FUNCTION_BLOCK CM_Sensor2State
VAR_INPUT
	PI_ManualMode : BOOL;
	PI_AutoMode : BOOL;
	
	PI_HMI_HAND : BOOL;
	PI_HMI_HAND_ON : BOOL;
	
	PI_Manual_ON : BOOL;
	PI_AutoHigh : BOOL;
	
	PI_AlarmHighEnable : BOOL;
	PI_AlarmLowEnable : BOOL;
	PI_Alarmdelay_H : DINT;
	PI_Alarmdelay_L : DINT;
	
	PI_Alarm_Condition_H : BOOL;
	PI_Alarm_Condition_L : BOOL;
	
	
	
END_VAR
VAR_OUTPUT
	PO_HMI_HAND : BOOL;
	PO_Manual : BOOL;
	PO_High : BOOL;
	
	PO_Alarm_H : BOOL;
	PO_Alarm_L : BOOL;
END_VAR
VAR
	Alarm_limit_Exceeded_H : BOOL;
	Alarm_limit_Exceeded_L : BOOL;
	
	prg_scan_H : DINT; // used for alarm delay
	prg_scan_L : DINT; // used for alarm delay
	
	Alarm_Ack_H : BOOL;
	Alarm_Ack_L : BOOL;
	
	alarmDelay_H : systemTimeDelay;
	alarmDelay_L : systemTimeDelay;
END_VAR
VAR_IN_OUT
	CM_UDT_CTRL : Udt_CM_Sensor2State;
	Plant_control : Udt_PlantControl;
END_VAR
VAR // added by the converter: edge detectors and wires of the graphical bodies
    _w1, _w2 : BOOL;
END_VAR

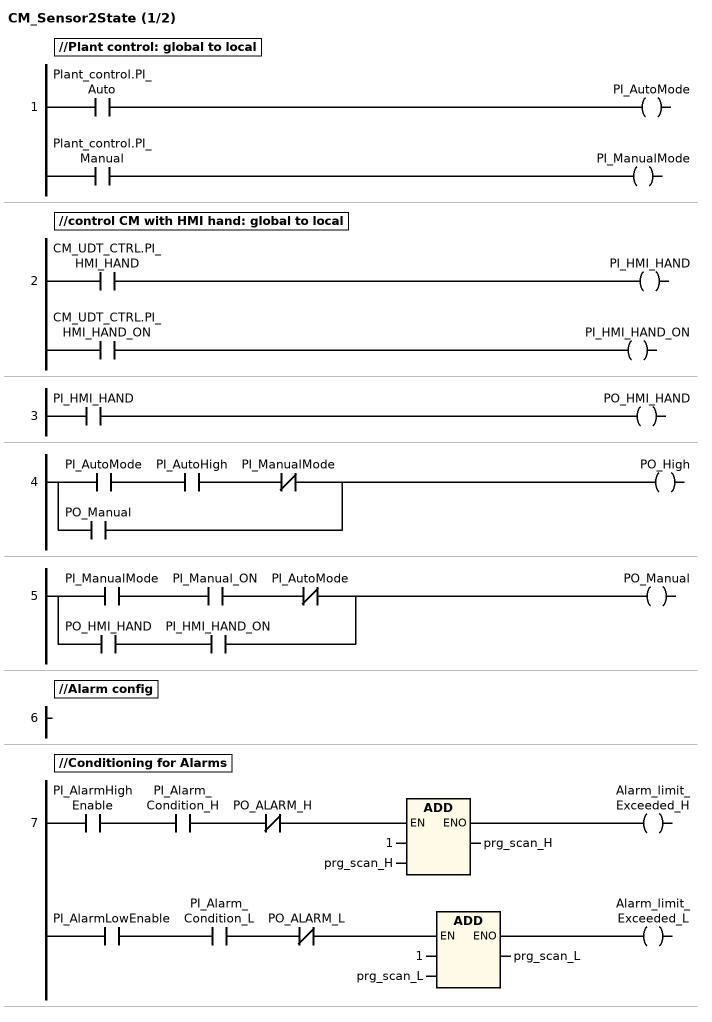
// NETWORK 1
// label: //Plant control: global to local
PI_AutoMode := Plant_control.PI_Auto;
PI_ManualMode := Plant_control.PI_Manual;

// NETWORK 2
// label: //control CM with HMI hand: global to local
PI_HMI_HAND := CM_UDT_CTRL.PI_HMI_HAND;
PI_HMI_HAND_ON := CM_UDT_CTRL.PI_HMI_HAND_ON;

// NETWORK 3
PO_HMI_HAND := PI_HMI_HAND;

// NETWORK 4
PO_High := PI_AutoMode AND PI_AutoHigh AND NOT PI_ManualMode OR PO_Manual;

// NETWORK 5
PO_Manual := PI_ManualMode AND PI_Manual_ON AND NOT PI_AutoMode OR PO_HMI_HAND AND PI_HMI_HAND_ON;

// NETWORK 6
// label: //Alarm config

// NETWORK 7
// label: //Conditioning for Alarms
_w1 := PI_AlarmHighEnable AND PI_Alarm_Condition_H AND NOT PO_ALARM_H;
IF _w1 THEN prg_scan_H := 1 + prg_scan_H; END_IF
Alarm_limit_Exceeded_H := _w1;
_w2 := PI_AlarmLowEnable AND PI_Alarm_Condition_L AND NOT PO_ALARM_L;
IF _w2 THEN prg_scan_L := 1 + prg_scan_L; END_IF
Alarm_limit_Exceeded_L := _w2;

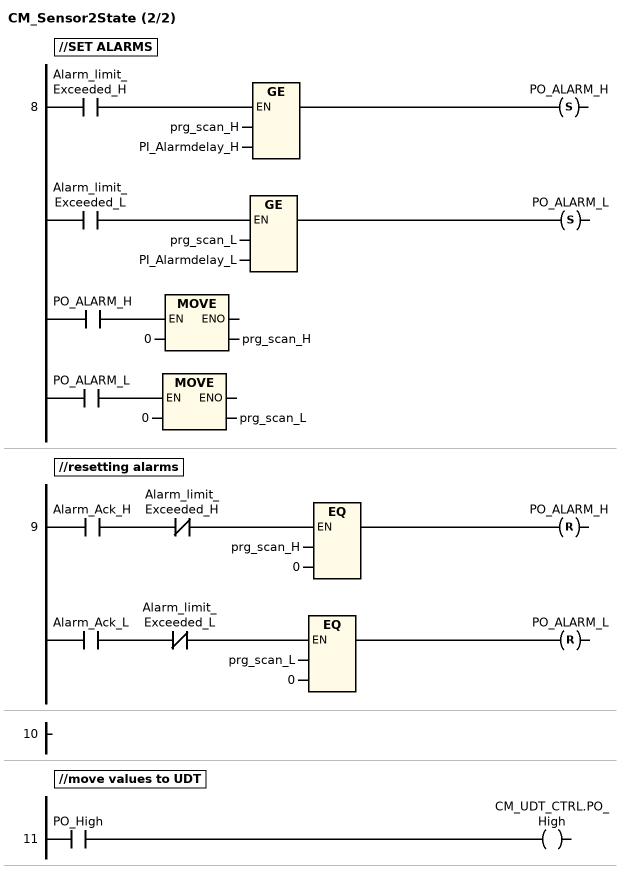
// NETWORK 8
// label: //SET ALARMS
PO_ALARM_H S= Alarm_limit_Exceeded_H AND prg_scan_H >= PI_Alarmdelay_H;
PO_ALARM_L S= Alarm_limit_Exceeded_L AND prg_scan_L >= PI_Alarmdelay_L;
IF PO_ALARM_H THEN prg_scan_H := 0; END_IF
IF PO_ALARM_L THEN prg_scan_L := 0; END_IF

// NETWORK 9
// label: //resetting alarms
PO_ALARM_H R= Alarm_Ack_H AND NOT Alarm_limit_Exceeded_H AND prg_scan_H = 0;
PO_ALARM_L R= Alarm_Ack_L AND NOT Alarm_limit_Exceeded_L AND prg_scan_L = 0;

// NETWORK 10

// NETWORK 11
// label: //move values to UDT
CM_UDT_CTRL.PO_High := PO_High;

END_FUNCTION_BLOCK

(* stored: Version 1.1.0.1, ProductVersion 3.1.4024.13
   POU CM_Sensor2State: Id {2164682c-c1a3-4d8d-bda6-2e325ad7b254}, SpecialFunc None *)
